(* LS Electric XG5000 project: CTD *)
(* PLC LSPLC *)
(* module base 0 slot 0: 입력 모듈:XGI-D22A/B (DC 24V 입력, 16점 (전류소스 싱크공용/ 전류소스 입력)) *)
(* module base 0 slot 1: 입력 모듈:XGI-D22A/B (DC 24V 입력, 16점 (전류소스 싱크공용/ 전류소스 입력)) *)
(* module base 0 slot 2: 출력 모듈:XGQ-RY2A/B (릴레이 출력, 16점 (2A용, Varistor 없음/Varistor 부착)) *)
(* module base 0 slot 3: 출력 모듈:XGQ-RY2A/B (릴레이 출력, 16점 (2A용, Varistor 없음/Varistor 부착)) *)

PROGRAM NewProgram (* task: 스캔 프로그램 *)
VAR
    C1 : CTD_INT;
    D1 : TIME;
    P0 : BOOL;
    T1 : TON;
    T2 : TON;
    이순신 : BOOL;
END_VAR

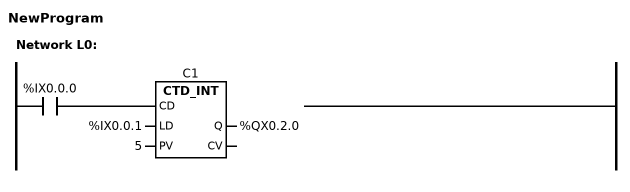
(* Rung L0 *)
C1(CD := %IX0.0.0, LD := %IX0.0.1, PV := 5, Q => %QX0.2.0);
END_PROGRAM